PROGRAM ChargeTime
VAR

	lca_charge_cal	 : ARRAY [1..6] OF LCA_CAL;
	i				 : INT := 1; // 1-8 instances
	j				 : INT := 1; //1 - 8 ch
	m				 : INT := 1;
	n				 : INT := 6; // no SR here yet
	a				 : INT := 1; 
	
	Q				 : REAL := 1; // Charge
	Current			 : REAL := 0.1; //100mA
	
	longestChargeTime: REAL;
	
END_VAR

//mapping hmi input to setpoints
FOR j := 1 TO n BY 1 DO	
	Setpoints.TDKLoad[j].TotalCapacitance	:= HMI_DB.TDKLoad[j].TotalCapacitance;
	Setpoints.TDKLoad[j].PSratedV 			:= HMI_DB.TDKLoad[j].PSratedV;
	Setpoints.TDKLoad[j].RequiredChargedV	:= HMI_DB.TDKLoad[j].RequiredChargedV;  
	Setpoints.TDKLoad[j].wLCA				:= HMI_DB.TDKLoad[j].wLCA;
	Setpoints.TDKLoad[j].NumOfCharger		:= HMI_DB.TDKLoad[j].NumOfCharger;	
	
	//charge time delay and elapse for HMI
	ChargeTime_DB.ChargeTimeStartDelay[j] := TIME_TO_INT((ChargeTime_DB.ChargerDelay_PT[j] - ChargeTime_DB.ChargerDelay_ET[j])/1000);
	ChargeTime_DB.ChargingTimeElapse[j] := TIME_TO_INT((ChargeTime_DB.ChargingTimeElapse_TON[j].PT - ChargeTime_DB.ChargingTimeElapse_TON[j].ET)/1000);
END_FOR

//ChargeTime_DB.PreFormChargeTimeStartDelay := TIME_TO_INT((ChargeTime_DB.PreFormChargeTime_PT - ChargeTime_DB.PreFormChargeTime_ET)/1000);
//ChargeTime_DB.PreFormChargingTimeElapse := TIME_TO_INT((ChargeTime_DB.PreFormChargingTimeElapse_TON.PT - ChargeTime_DB.PreFormChargingTimeElapse_TON.ET)/1000);

(*
//GLS 3
Setpoints.GLSLoad.TotalCapacitance	:= HMI_DB.GLSLoad.TotalCapacitance;
Setpoints.GLSLoad.PSratedV 			:= HMI_DB.GLSLoad.PSratedV;
//Setpoints.PreFormBank.RequiredChargedV	:= Recipe.PreFormBank.RequiredChargedV; //only thing that comes from the main plc recipe
//Setpoints.GLSLoad.wLCA				:= HMI_DB.GLSLoad.wLCA;
Setpoints.GLSLoad.NumOfCharger		:= HMI_DB.GLSLoad.NumOfCharger;	
*)


//veto
//this should not happen
FOR m := 1 TO n BY 1 DO
	IF Setpoints.TDKLoad[m].RequiredChargedV <= -2 THEN
		Setpoints.TDKLoad[m].RequiredChargedV := -2;
	END_IF	
END_FOR

(*
//charger 1 is 30kV*********************************************
IF 1000*(Setpoints.TDKLoad[1].RequiredChargedV) >= 12000 THEN
			Setpoints.TDKLoad[1].RequiredChargedV := (10000/1000); //limit at 10kv
			HMI_DB.TDKLoad[1].RequiredChargedV := (10000/1000);
	ELSIF Setpoints.TDKLoad[1].RequiredChargedV <= 0 THEN
			Setpoints.TDKLoad[1].RequiredChargedV := 0;
			HMI_DB.TDKLoad[1].RequiredChargedV := 0;
END_IF
//charger 1 is 30kV*********************************************
*)
//from 2 to 6
FOR i := 1 TO n BY 1 DO
	IF MCP_IO.Charger[i].ChargerType = E_ChargerType.TDK50kV THEN 
		//set limites of charger voltage input from HMI input
		IF 1000*(Setpoints.TDKLoad[i].RequiredChargedV) >= EngVal.UpperLimit50kVCaps THEN
			Setpoints.TDKLoad[i].RequiredChargedV := (EngVal.UpperLimit50kVCaps/1000); //limit at 35kv
			HMI_DB.TDKLoad[i].RequiredChargedV := (EngVal.UpperLimit50kVCaps/1000);
		ELSIF Setpoints.TDKLoad[i].RequiredChargedV <= 0 THEN
			Setpoints.TDKLoad[i].RequiredChargedV := 0;
			HMI_DB.TDKLoad[i].RequiredChargedV := 0;
		END_IF
	ELSIF MCP_IO.Charger[i].ChargerType = E_ChargerType.TDK12kV OR MCP_IO.Charger[i].ChargerType = E_ChargerType.TDK30kV THEN
		//set limites of charger voltage input from HMI input
		IF 1000*(Setpoints.TDKLoad[i].RequiredChargedV) >= EngVal.UpperLimit12kVCaps THEN
			Setpoints.TDKLoad[i].RequiredChargedV := (EngVal.UpperLimit12kVCaps/1000); //limit at 10kv
			HMI_DB.TDKLoad[i].RequiredChargedV := (EngVal.UpperLimit12kVCaps/1000); //limit at 10kv
		ELSIF Setpoints.TDKLoad[i].RequiredChargedV <= 0 THEN
			Setpoints.TDKLoad[i].RequiredChargedV := ABS(Setpoints.TDKLoad[i].RequiredChargedV);
			HMI_DB.TDKLoad[i].RequiredChargedV := ABS(Setpoints.TDKLoad[i].RequiredChargedV);
		END_IF
	END_IF;
END_FOR;
(*//ch 1 - 3
IF Setpoints.TDKLoad[1].RequiredChargedV >= 10 THEN
	Setpoints.TDKLoad[1].RequiredChargedV := 10;
	ELSIF Setpoints.TDKLoad[1].RequiredChargedV < 0 THEN
		Setpoints.TDKLoad[1].RequiredChargedV := ABS(Setpoints.TDKLoad[1].RequiredChargedV); 
END_IF
IF Setpoints.TDKLoad[2].RequiredChargedV >= 10 THEN
	Setpoints.TDKLoad[2].RequiredChargedV := 10;
	ELSIF Setpoints.TDKLoad[2].RequiredChargedV < 0 THEN
		Setpoints.TDKLoad[2].RequiredChargedV := ABS(Setpoints.TDKLoad[2].RequiredChargedV); 	
END_IF
IF Setpoints.TDKLoad[3].RequiredChargedV >= 10 THEN
	Setpoints.TDKLoad[3].RequiredChargedV := 10;
	ELSIF Setpoints.TDKLoad[3].RequiredChargedV < 0 THEN
		Setpoints.TDKLoad[3].RequiredChargedV := ABS(Setpoints.TDKLoad[3].RequiredChargedV); 	
END_IF

//ch 4-6
IF Setpoints.TDKLoad[4].RequiredChargedV >= 12 THEN
	Setpoints.TDKLoad[4].RequiredChargedV := 12;
	ELSIF Setpoints.TDKLoad[4].RequiredChargedV < 0 THEN
		Setpoints.TDKLoad[4].RequiredChargedV := ABS(Setpoints.TDKLoad[4].RequiredChargedV); 	
END_IF
IF Setpoints.TDKLoad[5].RequiredChargedV >= 12 THEN
	Setpoints.TDKLoad[5].RequiredChargedV := 12;
	ELSIF Setpoints.TDKLoad[5].RequiredChargedV < 0 THEN
		Setpoints.TDKLoad[5].RequiredChargedV := ABS(Setpoints.TDKLoad[5].RequiredChargedV); 	
END_IF
IF Setpoints.TDKLoad[6].RequiredChargedV >= 12 THEN
	Setpoints.TDKLoad[6].RequiredChargedV := 12;
	ELSIF Setpoints.TDKLoad[6].RequiredChargedV < 0 THEN
		Setpoints.TDKLoad[6].RequiredChargedV := ABS(Setpoints.TDKLoad[6].RequiredChargedV); 	
END_IF
*)

//chg time
FOR i := 1 TO n BY 1 DO
	lca_charge_cal[i](	PSratedV := Setpoints.TDKLoad[i].PSratedV, 
						RequiredChargeV := Setpoints.TDKLoad[i].RequiredChargedV, 
						LoadCapacitance := Setpoints.TDKLoad[i].TotalCapacitance, 
						NumOfCharger := Setpoints.TDKLoad[i].NumOfCharger, 
						wLCA := Setpoints.TDKLoad[i].wLCA
						);

	MCP_IO.Charger[i].ChargeTime.timeToChargeLoad := lca_charge_cal[i].TimeToChargeLoad;
	MCP_IO.Charger[i].ChargeTime.Power := lca_charge_cal[i].RespectedPower;
	
	IF Setpoints.TDKLoad[i].RequiredChargedV = 0 THEN
		MCP_IO.Charger[i].ChargeTime.timeToChargeLoad := 0;
		MCP_IO.Charger[i].ChargeTime.Power := 0;
	END_IF
END_FOR



(*
//gls - gls3 is preform cap charger
Q := 1000* Setpoints.GLSLoad.RequiredChargedV * (Setpoints.GLSLoad.TotalCapacitance / 1000000);
MCP_IO.GLS3_Load.timeToChargeLoad := Q / Current;
MCP_IO.GLS3_Load.Power := 1000*Setpoints.GLSLoad.RequiredChargedV * Current;
*)
//find the longest charge time.  //need more work
longestChargeTime := MAX( MCP_IO.Charger[1].ChargeTime.timeToChargeLoad,
							MCP_IO.Charger[2].ChargeTime.timeToChargeLoad,
							MCP_IO.Charger[3].ChargeTime.timeToChargeLoad,
							MCP_IO.Charger[4].ChargeTime.timeToChargeLoad,
							MCP_IO.Charger[5].ChargeTime.timeToChargeLoad,
							MCP_IO.Charger[6].ChargeTime.timeToChargeLoad,
							//MCP_IO.Charger[7].ChargeTime.timeToChargeLoad, //no SR yet
							GVL.pfcChargeTime
							(*MCP_IO.Charger[7].ChargeTime.timeToChargeLoad,
							MCP_IO.Charger[8].ChargeTime.timeToChargeLoad, *)
							(*MCP_IO.GLS3_Load.timeToChargeLoad*));

ChargeTime_DB.LongestChargeTime_PT := REAL_TO_TIME (1000*longestChargeTime);

//FOR a := 1 TO 8 BY 1 DO
FOR a := 1 TO n BY 1 DO
	IF (longestChargeTime - MCP_IO.Charger[a].ChargeTime.timeToChargeLoad) >= 0 THEN
		ChargeTime_DB.ChargerDelay_PT[a] := REAL_TO_TIME (1000*(longestChargeTime - MCP_IO.Charger[a].ChargeTime.timeToChargeLoad));
		ELSE 
			ChargeTime_DB.ChargerDelay_PT[a] := REAL_TO_TIME (1000*(MCP_IO.Charger[a].ChargeTime.timeToChargeLoad - longestChargeTime));
	END_IF;		

	//IF (longestChargeTime - MCP_IO.Charger[a+3].ChargeTime.timeToChargeLoad) >= 0 THEN
	//	ChargeTime_DB.SustChargeTime_PT[a] := REAL_TO_TIME (1000*(longestChargeTime - MCP_IO.Charger[a+3].ChargeTime.timeToChargeLoad));	
	//END_IF;	
	
END_FOR;

		
IF (longestChargeTime - GVL.pfcChargeTime)>= 0 THEN 
	ChargeTime_DB.pfcChargerDelay_PT := REAL_TO_TIME (1000*(longestChargeTime - GVL.pfcChargeTime));
	ELSE
		ChargeTime_DB.pfcChargerDelay_PT := REAL_TO_TIME (1000*(GVL.pfcChargeTime - longestChargeTime));	
END_IF

(*IF (longestChargeTime - MCP_IO.Charger[7].ChargeTime.timeToChargeLoad) >= 0 THEN
	ChargeTime_DB.FormChargeTime_PT[1] := REAL_TO_TIME (1000*(longestChargeTime - MCP_IO.Charger[7].ChargeTime.timeToChargeLoad));	
END_IF;	
IF (longestChargeTime - MCP_IO.Charger[8].ChargeTime.timeToChargeLoad) >= 0 THEN
	ChargeTime_DB.FormChargeTime_PT[2] := REAL_TO_TIME (1000*(longestChargeTime - MCP_IO.Charger[8].ChargeTime.timeToChargeLoad));	
END_IF;	

IF (longestChargeTime - MCP_IO.GLS3_Load.timeToChargeLoad) >= 0 THEN
		ChargeTime_DB.PreFormChargeTime_PT := REAL_TO_TIME (1000*(longestChargeTime - MCP_IO.GLS3_Load.timeToChargeLoad));
		ELSE
			ChargeTime_DB.PreFormChargeTime_PT := REAL_TO_TIME (1000*(MCP_IO.GLS3_Load.timeToChargeLoad -longestChargeTime));
END_IF;
*)


//IF i > 8 THEN 
IF i > n THEN 
	i := 1;
END_IF

IF j > n THEN
	j := 1;
END_IF

IF m > n THEN
	m := 1;
END_IF

//IF a > 8 THEN
IF a > n THEN
	a := 1;
END_IF;

END_PROGRAM

(* stored: Version 1.1.0.1, ProductVersion 3.1.4024.11
   POU ChargeTime: Id {28824270-3930-44b7-bfe2-d4b07042cd6b}, SpecialFunc None *)
